// TIA Portal V19 export
ORGANIZATION_BLOCK "Main"   // OB1, LAD, ProgramCycle
TITLE = "Main Program Sweep (Cycle)"
{ S7_Optimized_Access := 'TRUE' }
// stored: SetENOAutomatically false
   VAR_INPUT
      Initial_Call : Bool;   // Initial call of this OB
      Remanence : Bool;   // =True, if remanent data are available
   END_VAR
BEGIN

REGION Network 1
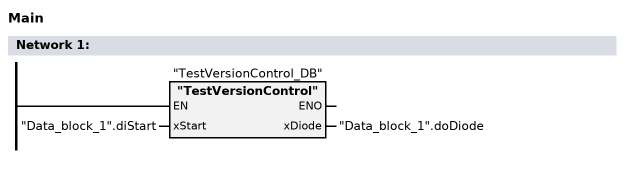
   RUNG wire#powerrail
      "TestVersionControl_DB"(xStart := "Data_block_1".diStart, xDiode => "Data_block_1".doDiode)
   END_RUNG
   // the same network as SCL:
   "TestVersionControl_DB"(xStart := "Data_block_1".diStart, xDiode => "Data_block_1".doDiode);   // "TestVersionControl"
END_REGION
END_ORGANIZATION_BLOCK
